TYPE ST_OutputTransportConfiguration :
STRUCT
	{attribute 'OPC.UA.DA.Description' := 'Dummy (for making struct visible on OPC UA'}
	Dummy						: BOOL;

END_STRUCT
END_TYPE

(* stored: Version 1.1.0.1, ProductVersion 3.1.4024.5
   DUT ST_OutputTransportConfiguration: Id {dac3ac19-63bc-41a4-93cc-754cd3d3252e} *)
